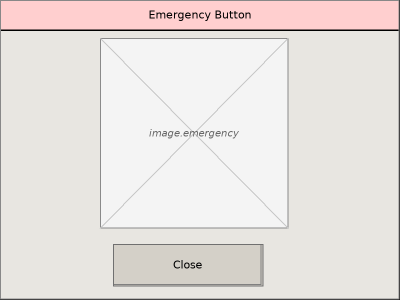
VISUALIZATION Popup  // 400x300
    Rectangle (0,0 400x30), "Emergency Button"
    Rectangle (0,30 400x270)
    Image (100,38 188x190), image: image.emergency
    Button (113,244 150x42), "Close"
        OnMouseClick: CloseDialog Dialog=Popup, Result=OK, NumpadKeypadSet=True
END_VISUALIZATION

(* stored: Version 1.1.0.1, ProductVersion 3.1.4024.12
   Visu Popup: Id {9271ba44-2e74-4701-a844-ede18adb2345} *)
